// TwinCAT 3 PLC project SerialComm_Library
// Title: SerialCom_Lib
// Company: Chua Siang Poh
// Author: Chua Siang Poh
// ProjectVersion: 2.0.1
// Description: Device library designed for simpler and modular serial communication applications in TwinCAT. Number of serial com channels can be specified in the Parameter list.
// ProgramVersion: 3.1.4020.10
// libraries:
//   Tc2_SerialCom, * (Beckhoff Automation GmbH)
//   Tc2_Standard, * (Beckhoff Automation GmbH)
//   Tc2_System, * (Beckhoff Automation GmbH)
//   Tc3_Interfaces, * (Beckhoff Automation GmbH)
//   Tc3_Module, * (Beckhoff Automation GmbH)
// project tree:
//   Base Component/Class/Common Base/ C_SERIALCOMM_PORT.TcPOU (not stored)
//   Base Component/Class/ C_SERIALCOMM_EL6.TcPOU (not stored), C_SERIALCOMM_PC.TcPOU (not stored)
//   Base Component/Interfaces/ I_SERIALCONTROLLER.TcIO
//   Version/ Global_Version.TcGVL (not stored)
// (motion and I/O tree: see PLC project motion_library)
// real-time tasks:
//   TASK PlcTask: cycle T#10ms, priority 20, ADS port 350

// ---- Base Component/Interfaces/I_SERIALCONTROLLER.TcIO
INTERFACE I_SERIALCONTROLLER

METHOD RECEIVE : DINT
VAR_INPUT
	ptr_data 	: PVOID;
END_VAR
VAR
END_VAR
END_METHOD

PROPERTY TIMEOUT : TIME
GET
END_GET
SET
END_SET
END_PROPERTY

METHOD SEND : DINT
VAR_INPUT
	ptr_data 	: PVOID;
	length		: UDINT;
END_VAR
END_METHOD

PROPERTY RECEIVE_PREFIX : STRING(15)
SET
END_SET
GET
END_GET
END_PROPERTY

PROPERTY RECEIVE_SUFFIX : STRING(15)
SET
END_SET
GET
END_GET
END_PROPERTY

METHOD FastBackgroundTask : DINT
END_METHOD

END_INTERFACE
